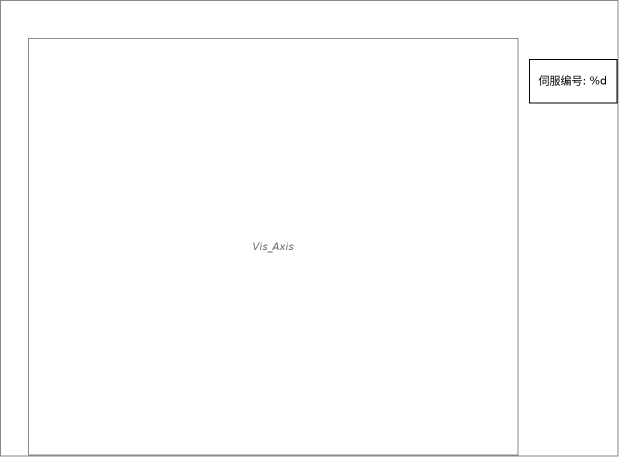
VISUALIZATION Vis_VirtualAxis  // 619x457
    Frame (28,38 490x417)
        shows Vis_Axis(Axis := MotionControl.Vis_VirtualAxisRef)
    Rectangle (529,59 88x44), "伺服编号: %d", text variable: MotionControl.Vis_VirtualAxisNoRef
        OnMouseClick: write the text variable via Default
END_VISUALIZATION

(* stored: Version 1.1.0.1, ProductVersion 3.1.4022.16
   Visu Vis_VirtualAxis: Id {ea1e71ae-5e65-448f-b2f9-603dbcd19d98} *)
